TYPE typeMotionRecordRow :
STRUCT
	Advanced:ULINT; //number of advanced
	Returned:ULINT; //number of returned
	stnPosnInput:STRING; //input value 
END_STRUCT
END_TYPE

(* stored: Version 1.1.0.1, ProductVersion 3.1.4024.11
   DUT typeMotionRecordRow: Id {f0495a16-7041-4694-9a4b-791fb5041a6e} *)
